// TIA Portal V19 export
VAR_GLOBAL   // PLC tag table "D03"
   D03_Ls AT %I1020.2 : Bool;   // 102DI2 - 190SQ2
END_VAR
